// TIA Portal V21 export
VAR_GLOBAL   // PLC tag table "K_Passo_Lavaggio_SterilizzatoreTubo"
END_VAR
VAR_GLOBAL CONSTANT   // user constants
   K_Passo_Risciacquo : Int := 1;
   K_Passo_Soda : Int := 2;
   K_Passo_RisciacquoSoda : Int := 3;
   K_Passo_Acido : Int := 4;
   K_Passo_RisciacquoAcido : Int := 5;
   K_Passo_Drenaggio : Int := 6;
END_VAR
